(* CODESYS project plc_chalet_base.library
   Title: CHALET_BaseComponents
   Version: 1.7.3
   Placeholder: CHALET_BaseComponents
   Company: Beckhoff CH

Project tree, tasks and I/O mapping:
  libraries: Tc2_Standard, 3.3.3.0 (Beckhoff Automation GmbH); Tc2_System, 3.4.25.0 (Beckhoff Automation GmbH); Tc2_Utilities, 3.3.52.0 (Beckhoff Automation GmbH); Tc3_EventLogger, 3.1.30.0 (Beckhoff Automation GmbH); Tc3_Module, 3.3.21.0 (Beckhoff Automation GmbH)
  COMPONENTs/
    Feedback/
      function block FB_CH_Feedback [ST]: ActiveCommand, Busy, Done, Error, ErrorId, HR, LastCommandAccepted
      interface I_CH_Feedback: ActiveCommand, Busy, Done, Error, ErrorId, HR, LastCommandAccepted
    HR/
      function CheckNotOk [ST]
      function CheckOk [ST]
      function GetMostSignificant [ST]
    List/
      CD_CH_List
      function block FB_CH_List [ST]: FindLUID, FindOID, FindOIDString, ResetIterator, Clear, Duplicate, Initialize, IsEmpty, Size, Update, AddObject, FindObject, GetNextObject, GetRandomObject, HasNextObject, RemoveObject
      interface I_CH_LIST: FindLUID, FindOID, FindOIDString, GetNextObject, GetRandomObject, HasNextObject, IsEmpty, ResetIterator, Size
    Object/
      CD_CH_Object
      function block FB_CH_Object [ST]: FB_init, Initialize, LUID, OID, TaskIndex, Update
      interface I_CH_Object: Initialize, LUID, OID, Update
  global variables BaseParameterlist
  00000000-0000-0000-0000-000000000000|Disclaimer Standard DE R1006.pdf
  Disclaimer Standard DE R1006.pdf
*)

// BaseParameterlist
{attribute 'qualified_only'}
VAR_GLOBAL CONSTANT
	(*Maximum length of List*)
	MAX_OBJECTS 			: UINT := 100;
END_VAR

// COMPONENTs/Feedback/FB_CH_Feedback
FUNCTION_BLOCK FB_CH_Feedback IMPLEMENTS I_CH_Feedback
VAR
    {attribute 'hide'}
    _hr : HRESULT;
    {attribute 'hide'}
    _activeCommand : STRING;
    {attribute 'hide'}
    _lastCommandAccepted : BOOL;
END_VAR

{attribute 'monitoring' := 'call'}
PROPERTY ActiveCommand : STRING;
GET
ActiveCommand := THIS^._ActiveCommand;
END_GET
SET
THIS^._ActiveCommand 		:= ActiveCommand;
//THIS^._LastAcceptedCommand	:= TRUE;  // Removed in V1.1
END_SET
END_PROPERTY

{attribute 'monitoring' := 'call'}
PROPERTY Busy : BOOL
GET
Busy := (THIS^._hr = S_PENDING);
END_GET
SET
IF Busy THEN
	THIS^._hr := S_PENDING;
END_IF
END_SET
END_PROPERTY

{attribute 'monitoring' := 'call'}
PROPERTY Done : BOOL
GET
Done := NOT THIS^.Busy AND NOT THIS^.Error;
END_GET
SET
IF Done THEN
	THIS^._hr := S_OK;
END_IF
END_SET
END_PROPERTY

{attribute 'monitoring' := 'call'}
PROPERTY Error : BOOL
GET
Error := FAILED(THIS^._hr);
END_GET
END_PROPERTY

{attribute 'monitoring' := 'call'}
PROPERTY ErrorId : UDINT
GET
ErrorId := DWORD_TO_UDINT(DINT_TO_DWORD(THIS^._hr) AND 16#0000FFFF); //only return the last two byte with the error Id
END_GET
SET
IF ErrorId <> 0 THEN
	//Add the nummber 42 to the hr at an position who is allways empty. 
	IF (TO_DINT(16#80420000 + ErrorId) <> THIS^._hr) THEN
		THIS^._hr := TO_DINT(16#80420000 + ErrorId);
	END_IF
END_IF
END_SET
END_PROPERTY

{attribute 'monitoring' := 'call'}
PROPERTY HR : HRESULT
GET
HR := THIS^._hr;
END_GET
SET
THIS^._hr := HR;
END_SET
END_PROPERTY

{attribute 'monitoring' := 'call'}
PROPERTY LastCommandAccepted : BOOL
GET
LastCommandAccepted := THIS^._lastCommandAccepted;
END_GET
SET
THIS^._lastCommandAccepted := LastCommandAccepted;
END_SET
END_PROPERTY

END_FUNCTION_BLOCK

// COMPONENTs/Feedback/I_CH_Feedback
INTERFACE I_CH_Feedback

{attribute 'monitoring' := 'call'}
PROPERTY ActiveCommand : STRING;
GET
END_GET
END_PROPERTY

{attribute 'monitoring' := 'call'}
PROPERTY Busy : BOOL
GET
END_GET
END_PROPERTY

{attribute 'monitoring' := 'call'}
PROPERTY Done : BOOL
GET
END_GET
END_PROPERTY

{attribute 'monitoring' := 'call'}
PROPERTY Error : BOOL
GET
END_GET
END_PROPERTY

{attribute 'monitoring' := 'call'}
PROPERTY ErrorId : UDINT
GET
END_GET
END_PROPERTY

{attribute 'monitoring' := 'call'}
PROPERTY HR : HRESULT
GET
END_GET
END_PROPERTY

{attribute 'monitoring' := 'call'}
PROPERTY LastCommandAccepted : BOOL
GET
END_GET
END_PROPERTY

END_INTERFACE

// COMPONENTs/HR/CheckNotOk
FUNCTION CheckNotOk : BOOL
VAR_INPUT
	hr : HRESULT;
END_VAR

CheckNotOk := (hr <> S_OK);

END_FUNCTION

// COMPONENTs/HR/CheckOk
FUNCTION CheckOk : BOOL
VAR_INPUT
	hr : HRESULT;
END_VAR

CheckOk := (hr = S_OK);

END_FUNCTION

// COMPONENTs/HR/GetMostSignificant
(*
	Return the most significant HRESULT input (hr1 or hr2).
	Example: if hr1:= S_Pending and hr2 := S_OK, then return S_Pending 
	Priority:(Error(incl. code) > Error(empty code) > S_WATCHDOGTIMEOUT > S_PENDING > S_FALSE > S_OK)
*)
FUNCTION GetMostSignificant : HRESULT
VAR_INPUT
	hr1 : HRESULT; //top priority if both hr1 and hr2 have an error code return this
	hr2 : HRESULT; //second priority if both hr1 and hr2 have an error code return hr1
END_VAR

//hr1 has an Error(incl. errorcode) 
IF hr1.31 AND ((hr1 AND 16#FFF) > 0) THEN
	GetMostSignificant := hr1;

//hr2 has an Error(incl. errorcode) 
ELSIF hr2.31 AND ((hr2 AND 16#FFF) > 0) THEN
	GetMostSignificant := hr2;

//hr1 has an Error(empty errorcode)
ELSIF hr1.31 THEN
	GetMostSignificant := hr1;

//hr2 has an Error(empty errorcode)
ELSIF hr2.31 THEN
	GetMostSignificant := hr2;
	
//hr1 has a higher SUCCESS code than hr2. (S_WATCHDOGTIMEOUT > S_PENDING > S_FALSE > S_OK)
ELSIF hr1 >= hr2 THEN
	GetMostSignificant := hr1;

//hr2 has a higher SUCCESS code than hr1. (S_WATCHDOGTIMEOUT > S_PENDING > S_FALSE > S_OK)
ELSE 
	GetMostSignificant := hr2;	
	
END_IF

END_FUNCTION

// COMPONENTs/List/FB_CH_List
FUNCTION_BLOCK FB_CH_List IMPLEMENTS I_CH_LIST
VAR
	{attribute 'hide'}
	nChObjectCount			: UINT;
	{attribute 'hide'}
	nChObjectNext			: UINT;
	aiChObjects				: ARRAY [1..BaseParameterlist.MAX_OBJECTS] OF I_CH_Object;
END_VAR

METHOD PUBLIC FindLUID : I_CH_OBJECT
VAR_INPUT
	sLUID	: STRING;
END_VAR
VAR
	i : UINT;
END_VAR
FOR i := 1 TO BaseParameterlist.MAX_OBJECTS DO
	IF aiChObjects[i] <> 0 AND_THEN aiChObjects[i].LUID = sLUID THEN
		FindLUID := aiChObjects[i];
		EXIT;
	END_IF
END_FOR
END_METHOD

METHOD FindOID : I_CH_OBJECT
VAR_INPUT
	oOID	: OTCID;
END_VAR
VAR
	i : UINT;
END_VAR
FOR i := 1 TO BaseParameterlist.MAX_OBJECTS DO
	IF aiChObjects[i] <> 0 AND_THEN aiChObjects[i].OID = oOID THEN
		FindOID := aiChObjects[i];
		EXIT;
	END_IF
END_FOR
END_METHOD

METHOD FindOIDString : I_CH_OBJECT
VAR_INPUT
	sOID	: STRING;
END_VAR
VAR
	i : UINT;
END_VAR
FOR i := 1 TO BaseParameterlist.MAX_OBJECTS DO
	IF aiChObjects[i] <> 0 AND_THEN DWORD_TO_HEXSTR(TO_DWORD(aiChObjects[i].OID),0,FALSE) = sOID THEN
		FindOIDString := aiChObjects[i];
		EXIT;
	END_IF
END_FOR
END_METHOD

METHOD PUBLIC ResetIterator : BOOL
VAR_INPUT
END_VAR
nChObjectNext := 0;
END_METHOD

METHOD PUBLIC Clear : BOOL
VAR
	nIdx : UINT;
END_VAR
FOR nIdx := 1 TO BaseParameterlist.MAX_OBJECTS DO
	aiChObjects[nIdx] := NULL;
END_FOR

nChObjectCount	:= 0;
nChObjectNext	:= 0;
END_METHOD

METHOD Duplicate : BOOL
VAR_INPUT
	CopyFrom : I_CH_LIST;
END_VAR
THIS^.Clear();

// Invalide input
IF CopyFrom = 0 THEN
	Duplicate := FALSE;;
	RETURN;
END_IF

// This list is to small
IF CopyFrom.Size > BaseParameterlist.MAX_OBJECTS THEN
	Duplicate := FALSE;;
	RETURN;
END_IF



CopyFrom.ResetIterator();
WHILE CopyFrom.HasNextObject() DO
	THIS^.AddObject(CopyFrom.GetNextObject());
END_WHILE

Duplicate := TRUE;
END_METHOD

METHOD Initialize : HRESULT
VAR_INPUT
END_VAR
VAR
	hr : HRESULT;
	nLoopIndex : UINT;
END_VAR
//Check if not Empty
IF UINT_TO_BOOL(nChObjectCount) THEN
	
	//FOR each element
	FOR nLoopIndex := 1 TO nChObjectCount DO
		// DO Init
		hr := GetMostSignificant(hr, aiChObjects[nLoopIndex].Initialize());
	END_FOR
	
END_IF

Initialize := hr;
END_METHOD

{attribute 'monitoring':='call'}
PROPERTY PUBLIC IsEmpty : BOOL
GET
IsEmpty := nChObjectCount = 0;
END_GET
END_PROPERTY

{attribute 'monitoring':='call'}
PROPERTY PUBLIC Size : UINT
GET
Size := nChObjectCount;
END_GET
END_PROPERTY

METHOD Update : HRESULT
VAR
	hr : HRESULT;
	nLoopIndex : UINT;
END_VAR
//Check if not Empty
IF UINT_TO_BOOL(nChObjectCount) THEN
	
	//FOR each element
	FOR nLoopIndex := 1 TO nChObjectCount DO
		// DO Update
		hr := GetMostSignificant(hr, aiChObjects[nLoopIndex].Update());
	END_FOR
	
END_IF

Update := hr;
END_METHOD

METHOD PUBLIC AddObject : HRESULT
VAR_INPUT
	iChObject	: I_CH_Object;
END_VAR
IF nChObjectCount >= BaseParameterlist.MAX_OBJECTS THEN
	AddObject := S_FALSE;
	RETURN;
END_IF

IF iChObject = 0 THEN
	AddObject := S_FALSE;
	RETURN;
END_IF

nChObjectCount := nChObjectCount + 1;
aiChObjects[nChObjectCount] := iChObject;

AddObject := S_OK;
END_METHOD

METHOD PUBLIC FindObject : BOOL
VAR_INPUT
	iChObject	: I_CH_Object;
END_VAR
VAR
	i : UINT;
END_VAR
//Check if not Empty
IF UINT_TO_BOOL(nChObjectCount) THEN
	
	FOR i := 1 TO nChObjectCount DO
		IF aiChObjects[i] = iChObject THEN
			FindObject := TRUE;
			EXIT;
		END_IF
	END_FOR
	
END_IF
END_METHOD

METHOD PUBLIC GetNextObject : I_CH_Object
VAR_INPUT
END_VAR
nChObjectNext := nChObjectNext + 1;
GetNextObject := aiChObjects[nChObjectNext];
END_METHOD

METHOD GetRandomObject : I_CH_Object
VAR_INPUT
END_VAR

VAR_INST
	{attribute 'hide'}
	fbDRAN : DRAND;
END_VAR

VAR
	nRandomIndex : UINT;
END_VAR
//Check if not Empty
IF UINT_TO_BOOL(nChObjectCount) THEN
	// Generate number 0..1
	fbDRAN(Seed:= 42);
	
	// 1..Size   = ((0..1)*(Size-1))+1
	nRandomIndex := LREAL_TO_UINT(fbDRAN.Num * (nChObjectCount-1))+1;
	
	GetRandomObject := aiChObjects[nRandomIndex];
	
END_IF
END_METHOD

METHOD PUBLIC HasNextObject : BOOL
VAR_INPUT
END_VAR
HasNextObject := (nChObjectNext < nChObjectCount);
END_METHOD

METHOD PUBLIC RemoveObject : BOOL
VAR_INPUT
	iChObject	: I_CH_Object;
END_VAR

VAR
	nIdx			: UDINT;
END_VAR
RemoveObject := FALSE;

IF iChObject = 0 THEN
	RETURN;
END_IF

IF NOT THIS^.FindObject(iChObject) THEN
	RETURN;
END_IF

FOR nIdx := 1 TO BaseParameterlist.MAX_OBJECTS DO
	IF aiChObjects[nIdx] = iChObject THEN
		aiChObjects[nIdx] := NULL;	
		
		nChObjectCount := nChObjectCount - 1;
		
		// Fill up the empty slot
		MEMMOVE(ADR(aiChObjects[nIdx]), ADR(aiChObjects[nIdx + 1]), SIZEOF(aiChObjects[nIdx]) * (BaseParameterlist.MAX_OBJECTS - nIdx));
	
		RemoveObject := TRUE;
		EXIT;
	END_IF
END_FOR
END_METHOD

END_FUNCTION_BLOCK

// COMPONENTs/List/I_CH_LIST
INTERFACE I_CH_LIST

METHOD PUBLIC FindLUID : I_CH_OBJECT
VAR_INPUT
	sLUID	: STRING;
END_VAR
END_METHOD

METHOD FindOID : I_CH_OBJECT
VAR_INPUT
	oOID	: OTCID;
END_VAR
END_METHOD

METHOD FindOIDString : I_CH_OBJECT
VAR_INPUT
	sOID	: STRING;
END_VAR
END_METHOD

METHOD PUBLIC GetNextObject : I_CH_Object
VAR_INPUT
END_VAR
END_METHOD

METHOD GetRandomObject : I_CH_Object
VAR_INPUT
END_VAR
END_METHOD

METHOD PUBLIC HasNextObject : BOOL
VAR_INPUT
END_VAR
END_METHOD

{attribute 'monitoring':='call'}
PROPERTY PUBLIC IsEmpty : BOOL
GET
END_GET
END_PROPERTY

METHOD PUBLIC ResetIterator : BOOL
VAR_INPUT
END_VAR
END_METHOD

{attribute 'monitoring':='call'}
PROPERTY PUBLIC Size : UINT
GET
END_GET
END_PROPERTY

END_INTERFACE

// COMPONENTs/Object/I_CH_Object
INTERFACE I_CH_Object EXTENDS __SYSTEM.IQueryInterface

METHOD Initialize : HRESULT
END_METHOD

{attribute 'monitoring':='call'}
PROPERTY LUID : STRING
GET
END_GET
END_PROPERTY

{attribute 'monitoring':='call'}
PROPERTY OID : OTCID
GET
END_GET
END_PROPERTY

METHOD Update : HRESULT
VAR_INPUT
END_VAR
END_METHOD

END_INTERFACE

// COMPONENTs/Object/FB_CH_Object
FUNCTION_BLOCK FB_CH_Object IMPLEMENTS I_CH_Object
VAR
	fbSelf : FB_TcSourceInfo;
	
	{attribute 'hide'}
	nTaskIndex : BYTE; //Used in TwinCAT_SystemInfoVarList._TaskInfo
END_VAR

METHOD FB_init : BOOL
VAR_INPUT
	bInitRetains : BOOL; // if TRUE, the retain variables are initialized (warm start / cold start)
	bInCopyCode : BOOL;  // if TRUE, the instance afterwards gets moved into the copy code (online change)
END_VAR
VAR
	fbGetCurTaskIdx  : GETCURTASKINDEX;
END_VAR
fbGetCurTaskIdx();
THIS^.nTaskIndex := fbGetCurTaskIdx.index;
END_METHOD

METHOD Initialize : HRESULT
Initialize := S_OK;
END_METHOD

{attribute 'monitoring':='call'}
PROPERTY LUID : STRING
GET
LUID := THIS^.fbSelf.sName;
END_GET
END_PROPERTY

{attribute 'monitoring':='call'}
PROPERTY OID : OTCID
GET
OID := 0;
END_GET
END_PROPERTY

PROPERTY PROTECTED TaskIndex : BYTE //Used in TwinCAT_SystemInfoVarList._TaskInfo
GET
TaskIndex := THIS^.nTaskIndex;
END_GET
END_PROPERTY

METHOD Update : HRESULT
VAR_INPUT
END_VAR
Update := S_OK;
END_METHOD

END_FUNCTION_BLOCK
